// TIA Portal V17 export
// export: Created 2024-09-03T21:54:52.2531317Z, ExportSetting WithDefaults, DisplayName Totally Integrated Automation Portal, DisplayVersion V17 Update 7, DisplayName TIA Portal Openness, DisplayVersion V17 Update 7, DisplayName TIA Portal Version Control Interface, DisplayVersion V17, DisplayName SINAMICS Startdrive Advanced, DisplayVersion V17 SP2, DisplayName SINAMICS Startdrive G110M, G120, G120C, G120D, G120P, G115D, DisplayVersion V17 SP2, DisplayName SINAMICS Startdrive G130, G150, S120, S150, SINAMICS MV, S210, DisplayVersion V17 SP2, DisplayName STEP 7 Professional, DisplayVersion V17 Update 7, DisplayName STEP 7 Safety, DisplayVersion V17 Update 6, DisplayName WinCC Advanced / Unified PC, DisplayVersion V17 Update 7
DATA_BLOCK "READER_REAR_TUBE"   // DB76
VERSION : 0.1
// stored: AutoNumber true, DBAccessibleFromOPCUA true, DBAccessibleFromWebserver true, InstanceOfName READER_LOGIC, InstanceOfType FB
"READER_LOGIC"
   // VAR_INPUT
   //    MODE : UInt;
   //    INIT_SCAN : Bool;
   //    SCAN_BUSY : Bool;
   //    SCAN_COMPLETE : Bool;
   //    STA_REC_1 : Bool;
   //    STA_REC : Bool;
   //    SCAN_OK1 : Bool;
   //    SCAN_OK2 : Bool;
   //    IJC_DISABLE : Bool;
   //    SCAN_LABEL : String;
   //    SCAN_POSITION : Int;
   //    SCAN_LEN : Int;
   //    READ_OF_SCAN : HW_SUBMODULE;
   //    NUM_OF_TUBE : Bool;
   //    RESET_SCANER : Bool;
   // END_VAR
   // VAR_OUTPUT
   //    REQUEST_SCAN : Bool;
   //    READ_STRG : String;
   //    SCAN_OK : Bool;
   //    MSG_STATUS_REQ : Bool;
   //    NFP_AUX : String;
   //    LECTURA_SCANER_ST : String;
   //    SCAN_CLEAR : Bool;
   // END_VAR
   // VAR
   //    RET_TRIG : IEC_TIMER;
   // END_VAR
BEGIN
END_DATA_BLOCK
